// Mitsubishi GX Works2 project: Atividade1   PLC: Q03UDV
// input1_out1_m

PROGRAM MAIN
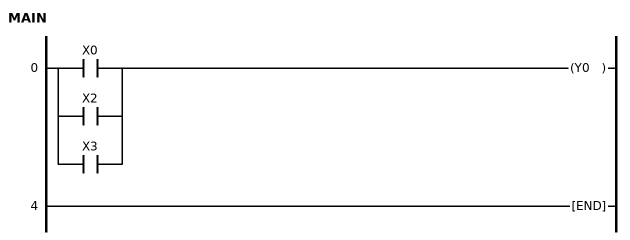
0     LD      X0
      OR      X2
      OR      X3
      OUT     Y0
4     END
END_PROGRAM
